// Mitsubishi GX Works2 project: 231002-001- exercicios-4   PLC: Q03UDV

// global labels: Global1
VAR_GLOBAL
  Up_Down AT M34 : BOOL;
END_VAR

// task Task_01 (event TRUE, interval 0, priority 31): POU_01

PROGRAM POU_01
VAR
  CTD_1 : CTD;
  CTU_1 : CTU;
  meuc : CTU;
  novo : CTUD;
  TP_1 : TP;
  TON_1 : TON;
  TOF_1 : TOF;
  dr : TIME;
  timetp : TIME;
  timeon : TIME;
  TimeOFF : TIME;
END_VAR
(* structured ladder/FBD written out as ST: instructions are called as NAME(EN, inputs, outputs); _pN, _eN, _tN stand for wires *)
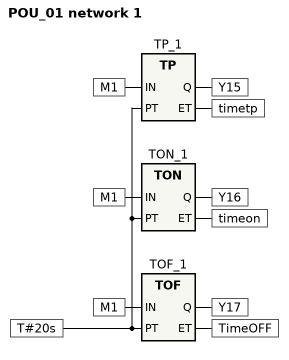
(* network 1 *)
TP_1(IN := M1, PT := T#20s, Q => Y15, ET => timetp);
TON_1(IN := M1, PT := T#20s, Q => Y16, ET => timeon);
TOF_1(IN := M1, PT := T#20s, Q => Y17, ET => TimeOFF);
END_PROGRAM
